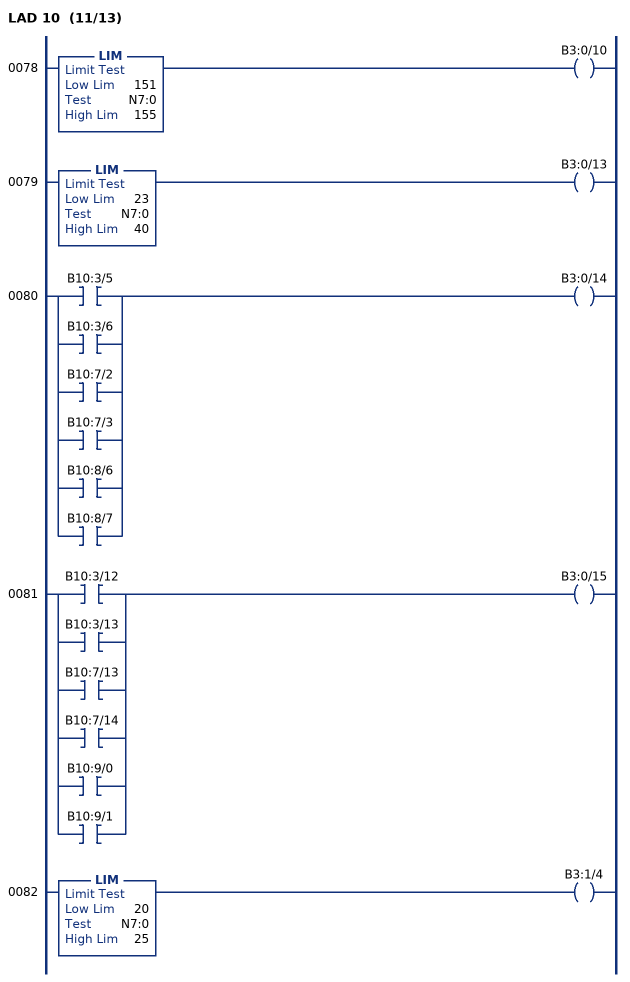
% Rung: 78 %
SOR LIM 151 N7:0 155 OTE B3:0/10 EOR
% Rung: 79 %
SOR LIM 23 N7:0 40 OTE B3:0/13 EOR
% Rung: 80 %
SOR BST XIC B10:3/5 NXB XIC B10:3/6 NXB XIC B10:7/2 NXB XIC B10:7/3 NXB XIC B10:8/6 NXB XIC B10:8/7 BND OTE B3:0/14 EOR
% Rung: 81 %
SOR BST XIC B10:3/12 NXB XIC B10:3/13 NXB XIC B10:7/13 NXB XIC B10:7/14 NXB XIC B10:9/0 NXB XIC B10:9/1 BND OTE B3:0/15 EOR
% Rung: 82 %
SOR LIM 20 N7:0 25 OTE B3:1/4 EOR

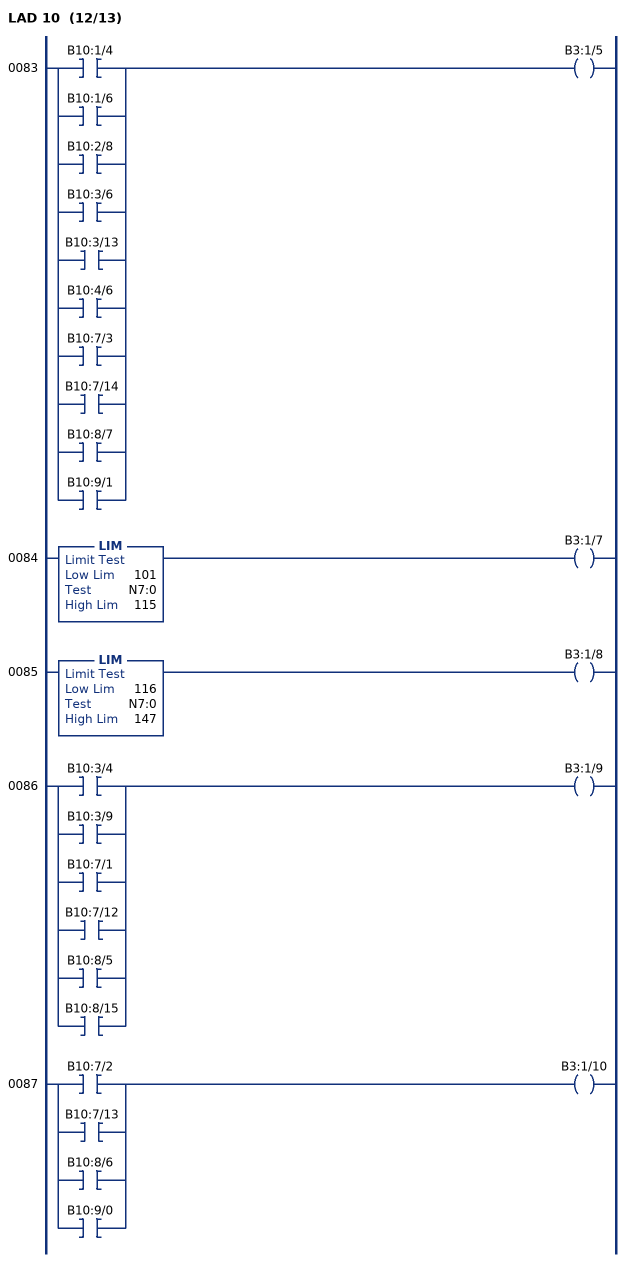
% Rung: 83 %
SOR BST XIC B10:1/4 NXB XIC B10:1/6 NXB XIC B10:2/8 NXB XIC B10:3/6 NXB XIC B10:3/13 NXB XIC B10:4/6 NXB XIC B10:7/3 NXB XIC B10:7/14 NXB XIC B10:8/7 NXB XIC B10:9/1 BND OTE B3:1/5 EOR
% Rung: 84 %
SOR LIM 101 N7:0 115 OTE B3:1/7 EOR
% Rung: 85 %
SOR LIM 116 N7:0 147 OTE B3:1/8 EOR
% Rung: 86 %
SOR BST XIC B10:3/4 NXB XIC B10:3/9 NXB XIC B10:7/1 NXB XIC B10:7/12 NXB XIC B10:8/5 NXB XIC B10:8/15 BND OTE B3:1/9 EOR
% Rung: 87 %
SOR BST XIC B10:7/2 NXB XIC B10:7/13 NXB XIC B10:8/6 NXB XIC B10:9/0 BND OTE B3:1/10 EOR

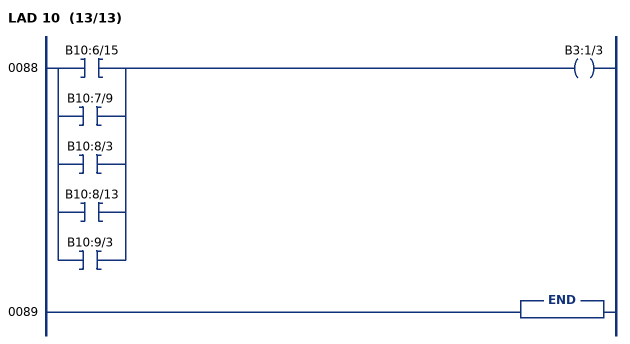
% Rung: 88 %
SOR BST XIC B10:6/15 NXB XIC B10:7/9 NXB XIC B10:8/3 NXB XIC B10:8/13 NXB XIC B10:9/3 BND OTE B3:1/3 EOR
% Rung: 89 %
SOR END EOR

LADDER 11
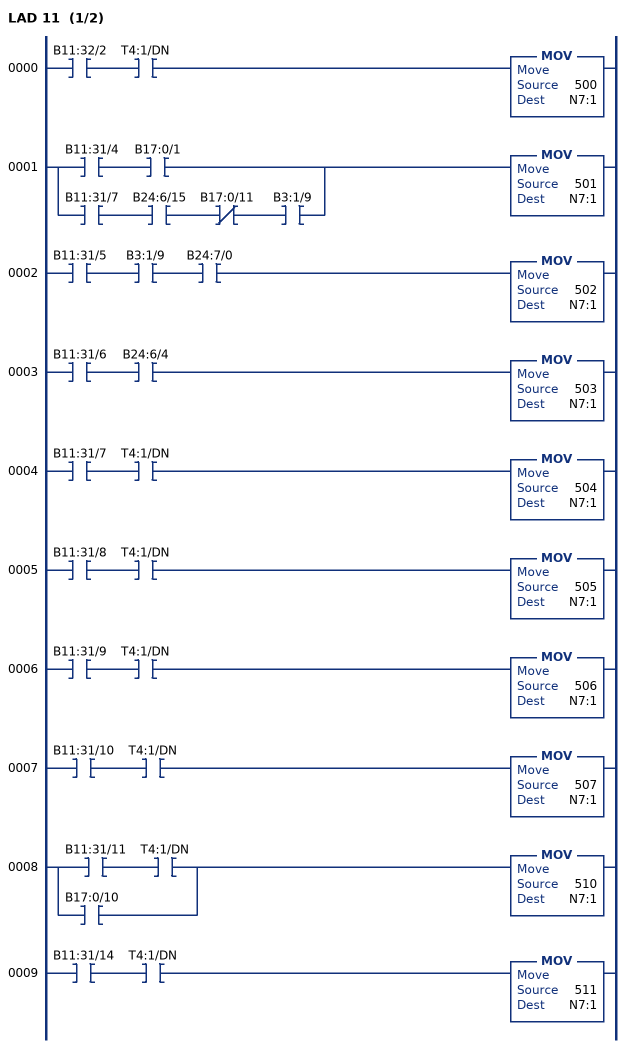
% Rung: 0 %
SOR XIC B11:32/2 XIC T4:1/DN MOV 500 N7:1 EOR
% Rung: 1 %
SOR BST XIC B11:31/4 XIC B17:0/1 NXB XIC B11:31/7 XIC B24:6/15 XIO B17:0/11 XIC B3:1/9 BND MOV 501 N7:1 EOR
% Rung: 2 %
SOR XIC B11:31/5 XIC B3:1/9 XIC B24:7/0 MOV 502 N7:1 EOR
% Rung: 3 %
SOR XIC B11:31/6 XIC B24:6/4 MOV 503 N7:1 EOR
% Rung: 4 %
SOR XIC B11:31/7 XIC T4:1/DN MOV 504 N7:1 EOR
% Rung: 5 %
SOR XIC B11:31/8 XIC T4:1/DN MOV 505 N7:1 EOR
% Rung: 6 %
SOR XIC B11:31/9 XIC T4:1/DN MOV 506 N7:1 EOR
% Rung: 7 %
SOR XIC B11:31/10 XIC T4:1/DN MOV 507 N7:1 EOR
% Rung: 8 %
SOR BST XIC B11:31/11 XIC T4:1/DN NXB XIC B17:0/10 BND MOV 510 N7:1 EOR
% Rung: 9 %
SOR XIC B11:31/14 XIC T4:1/DN MOV 511 N7:1 EOR

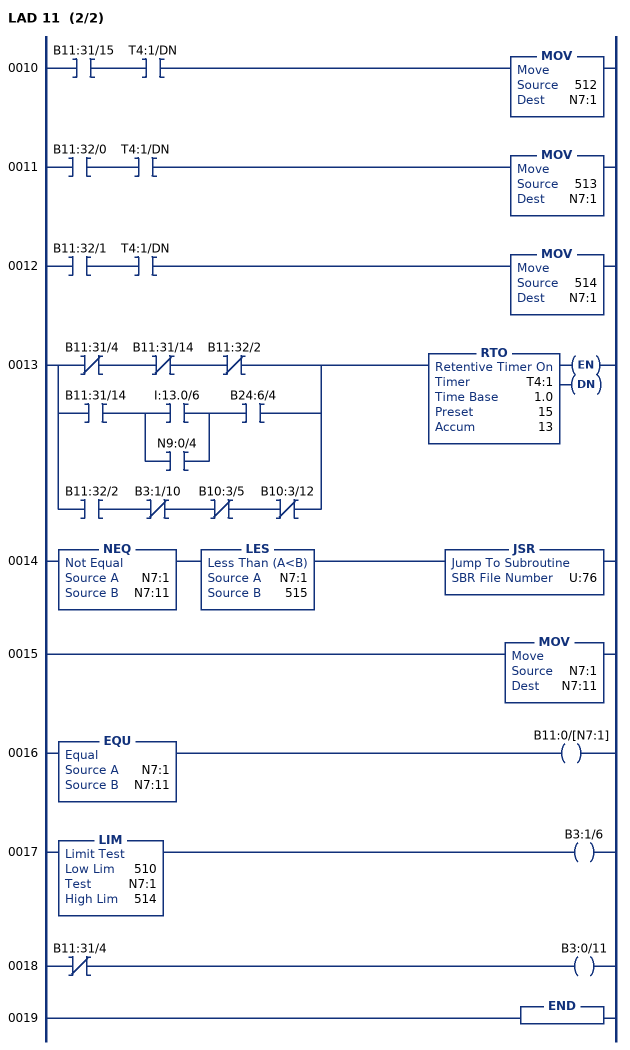
% Rung: 10 %
SOR XIC B11:31/15 XIC T4:1/DN MOV 512 N7:1 EOR
% Rung: 11 %
SOR XIC B11:32/0 XIC T4:1/DN MOV 513 N7:1 EOR
% Rung: 12 %
SOR XIC B11:32/1 XIC T4:1/DN MOV 514 N7:1 EOR
% Rung: 13 %
SOR BST XIO B11:31/4 XIO B11:31/14 XIO B11:32/2 NXB XIC B11:31/14 BST XIC I:13.0/6 NXB XIC N9:0/4 BND XIC B24:6/4 NXB XIC B11:32/2 XIO B3:1/10 XIO B10:3/5 XIO B10:3/12 BND RTO T4:1 1.0 15 13 EOR
% Rung: 14 %
SOR NEQ N7:1 N7:11 LES N7:1 515 JSR U:76 EOR
% Rung: 15 %
SOR MOV N7:1 N7:11 EOR
% Rung: 16 %
SOR EQU N7:1 N7:11 OTE B11:0/[N7:1] EOR
% Rung: 17 %
SOR LIM 510 N7:1 514 OTE B3:1/6 EOR
% Rung: 18 %
SOR XIO B11:31/4 OTE B3:0/11 EOR
% Rung: 19 %
SOR END EOR

LADDER 12
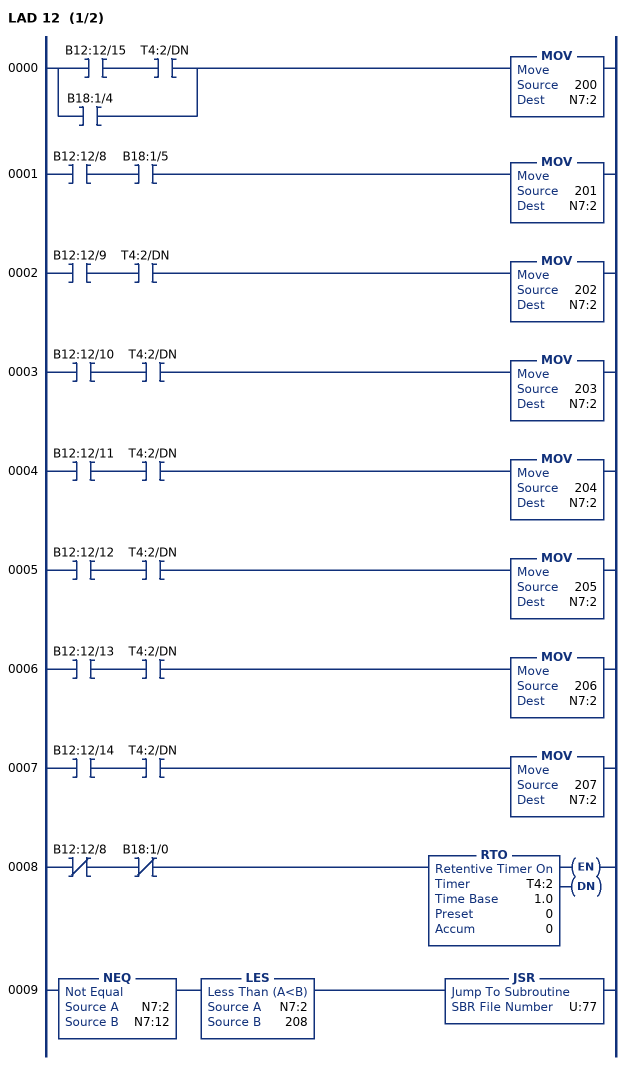
% Rung: 0 %
SOR BST XIC B12:12/15 XIC T4:2/DN NXB XIC B18:1/4 BND MOV 200 N7:2 EOR
% Rung: 1 %
SOR XIC B12:12/8 XIC B18:1/5 MOV 201 N7:2 EOR
% Rung: 2 %
SOR XIC B12:12/9 XIC T4:2/DN MOV 202 N7:2 EOR
% Rung: 3 %
SOR XIC B12:12/10 XIC T4:2/DN MOV 203 N7:2 EOR
% Rung: 4 %
SOR XIC B12:12/11 XIC T4:2/DN MOV 204 N7:2 EOR
% Rung: 5 %
SOR XIC B12:12/12 XIC T4:2/DN MOV 205 N7:2 EOR
% Rung: 6 %
SOR XIC B12:12/13 XIC T4:2/DN MOV 206 N7:2 EOR
% Rung: 7 %
SOR XIC B12:12/14 XIC T4:2/DN MOV 207 N7:2 EOR
% Rung: 8 %
SOR XIO B12:12/8 XIO B18:1/0 RTO T4:2 1.0 0 0 EOR
% Rung: 9 %
SOR NEQ N7:2 N7:12 LES N7:2 208 JSR U:77 EOR

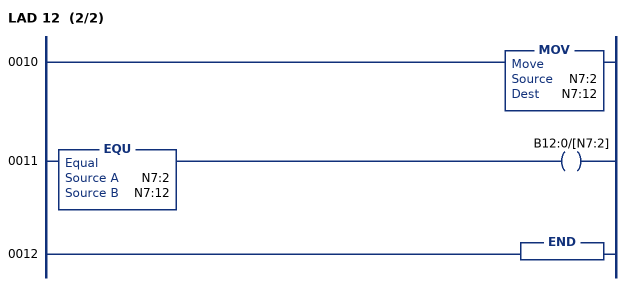
% Rung: 10 %
SOR MOV N7:2 N7:12 EOR
% Rung: 11 %
SOR EQU N7:2 N7:12 OTE B12:0/[N7:2] EOR
% Rung: 12 %
SOR END EOR

LADDER 15
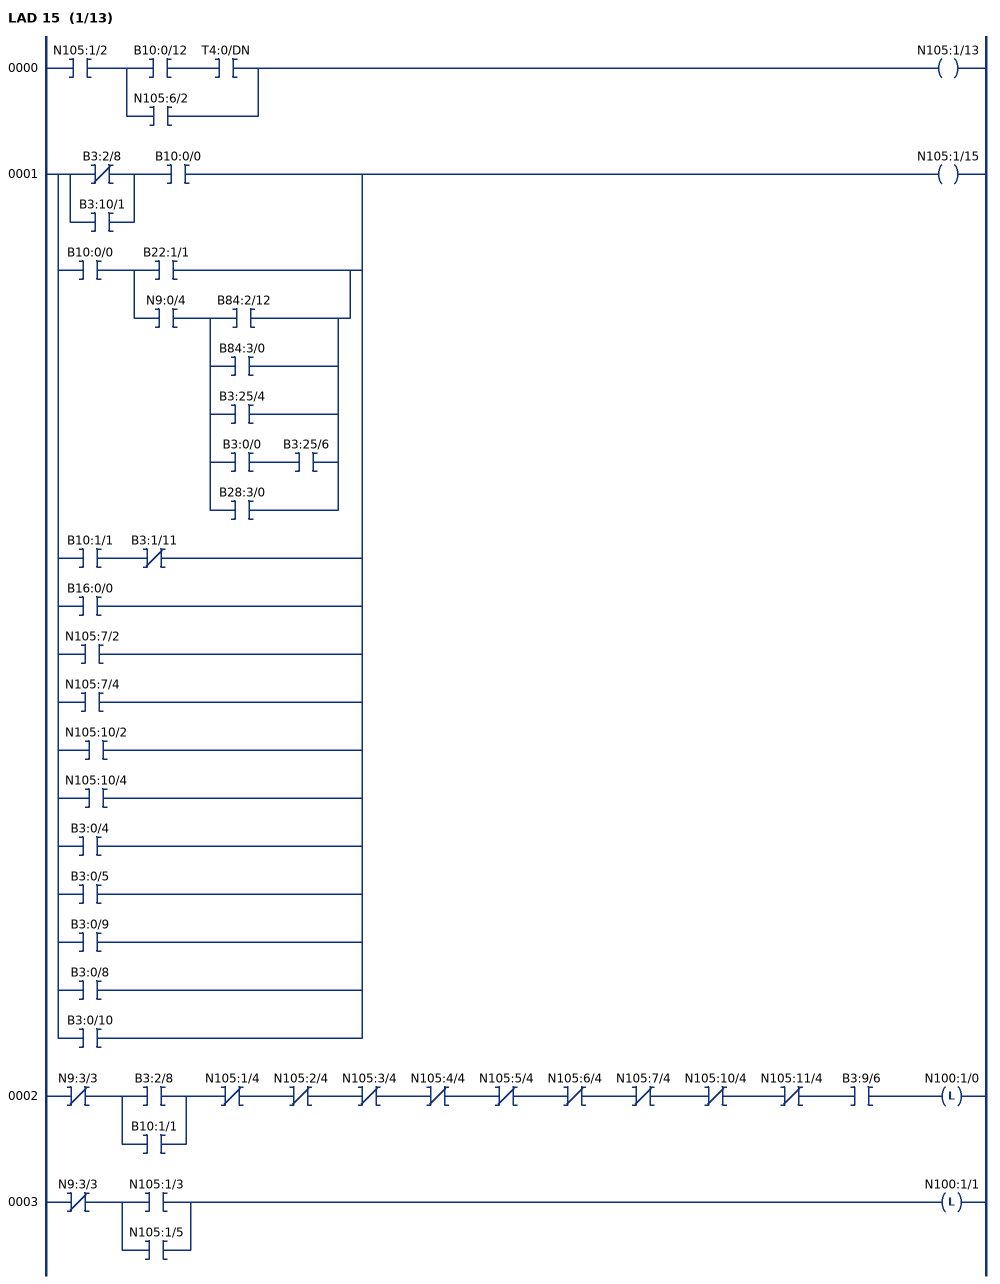
% Rung: 0 %
SOR XIC N105:1/2 BST XIC B10:0/12 XIC T4:0/DN NXB XIC N105:6/2 BND OTE N105:1/13 EOR
% Rung: 1 %
SOR BST BST XIO B3:2/8 NXB XIC B3:10/1 BND XIC B10:0/0 NXB XIC B10:0/0 BST XIC B22:1/1 NXB XIC N9:0/4 BST XIC B84:2/12 NXB XIC B84:3/0 NXB XIC B3:25/4 NXB XIC B3:0/0 XIC B3:25/6 NXB XIC B28:3/0 BND BND NXB XIC B10:1/1 XIO B3:1/11 NXB XIC B16:0/0 NXB XIC N105:7/2 NXB XIC N105:7/4 NXB XIC N105:10/2 NXB XIC N105:10/4 NXB XIC B3:0/4 NXB XIC B3:0/5 NXB XIC B3:0/9 NXB XIC B3:0/8 NXB XIC B3:0/10 BND OTE N105:1/15 EOR
% Rung: 2 %
SOR XIO N9:3/3 BST XIC B3:2/8 NXB XIC B10:1/1 BND XIO N105:1/4 XIO N105:2/4 XIO N105:3/4 XIO N105:4/4 XIO N105:5/4 XIO N105:6/4 XIO N105:7/4 XIO N105:10/4 XIO N105:11/4 XIC B3:9/6 OTL N100:1/0 EOR
% Rung: 3 %
SOR XIO N9:3/3 BST XIC N105:1/3 NXB XIC N105:1/5 BND OTL N100:1/1 EOR

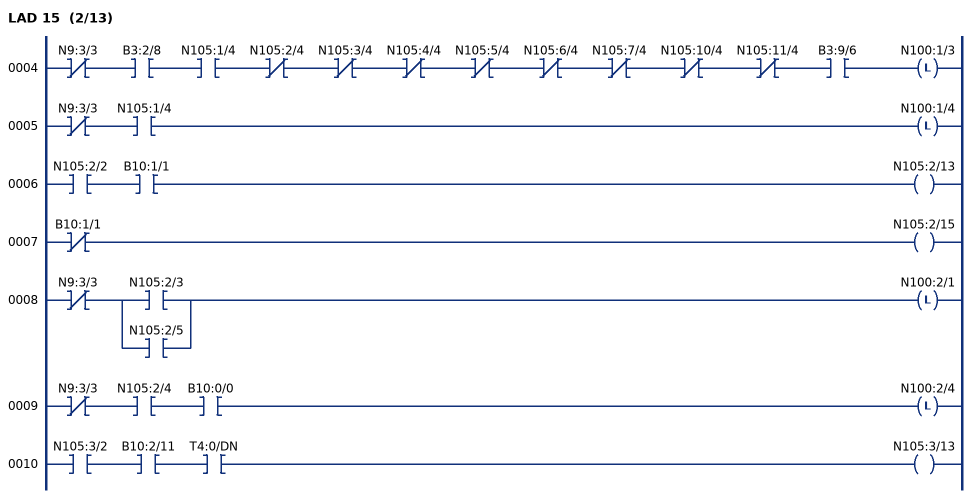
% Rung: 4 %
SOR XIO N9:3/3 XIC B3:2/8 XIC N105:1/4 XIO N105:2/4 XIO N105:3/4 XIO N105:4/4 XIO N105:5/4 XIO N105:6/4 XIO N105:7/4 XIO N105:10/4 XIO N105:11/4 XIC B3:9/6 OTL N100:1/3 EOR
% Rung: 5 %
SOR XIO N9:3/3 XIC N105:1/4 OTL N100:1/4 EOR
% Rung: 6 %
SOR XIC N105:2/2 XIC B10:1/1 OTE N105:2/13 EOR
% Rung: 7 %
SOR XIO B10:1/1 OTE N105:2/15 EOR
% Rung: 8 %
SOR XIO N9:3/3 BST XIC N105:2/3 NXB XIC N105:2/5 BND OTL N100:2/1 EOR
% Rung: 9 %
SOR XIO N9:3/3 XIC N105:2/4 XIC B10:0/0 OTL N100:2/4 EOR
% Rung: 10 %
SOR XIC N105:3/2 XIC B10:2/11 XIC T4:0/DN OTE N105:3/13 EOR

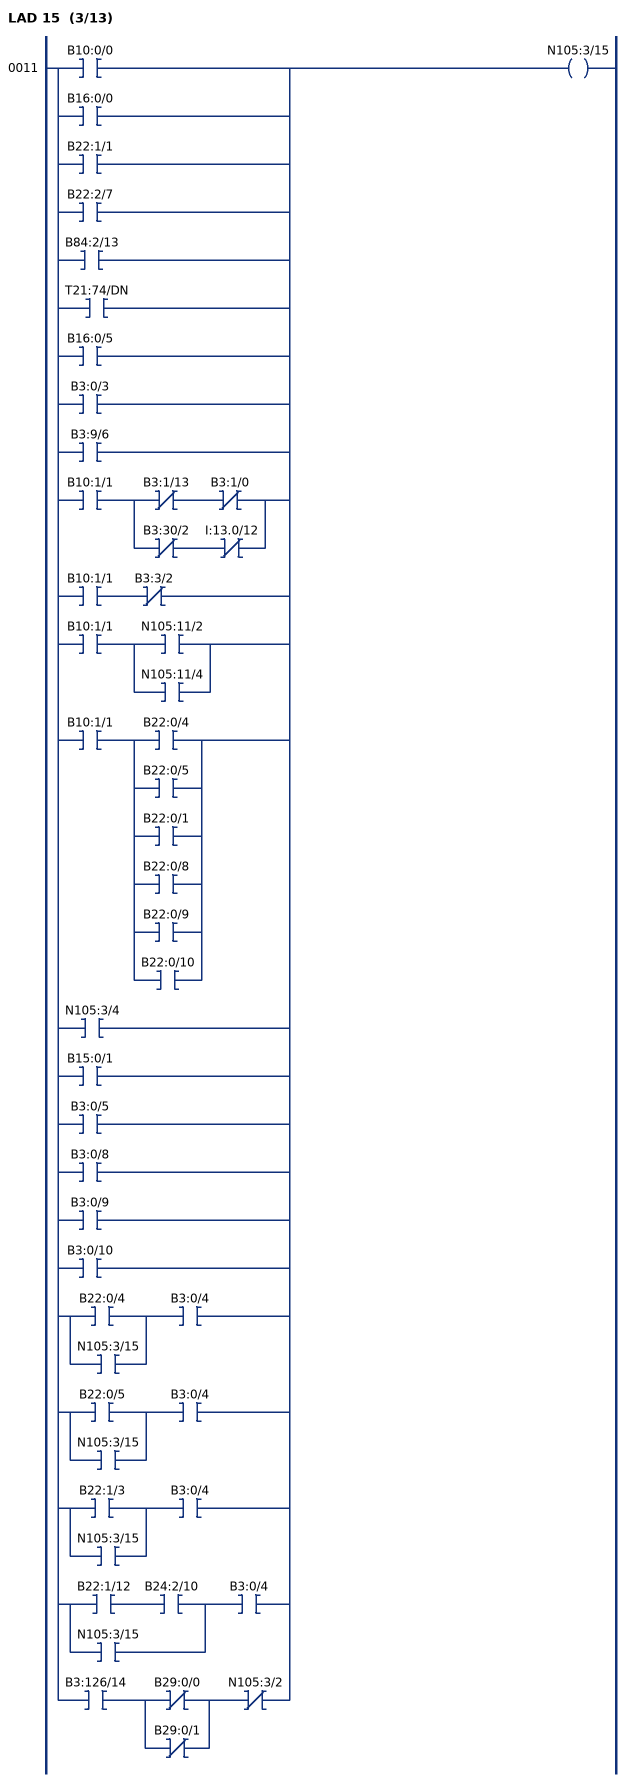
% Rung: 11 %
SOR BST XIC B10:0/0 NXB XIC B16:0/0 NXB XIC B22:1/1 NXB XIC B22:2/7 NXB XIC B84:2/13 NXB XIC T21:74/DN NXB XIC B16:0/5 NXB XIC B3:0/3 NXB XIC B3:9/6 NXB XIC B10:1/1 BST XIO B3:1/13 XIO B3:1/0 NXB XIO B3:30/2 XIO I:13.0/12 BND NXB XIC B10:1/1 XIO B3:3/2 NXB XIC B10:1/1 BST XIC N105:11/2 NXB XIC N105:11/4 BND NXB XIC B10:1/1 BST XIC B22:0/4 NXB XIC B22:0/5 NXB XIC B22:0/1 NXB XIC B22:0/8 NXB XIC B22:0/9 NXB XIC B22:0/10 BND NXB XIC N105:3/4 NXB XIC B15:0/1 NXB XIC B3:0/5 NXB XIC B3:0/8 NXB XIC B3:0/9 NXB XIC B3:0/10 NXB BST XIC B22:0/4 NXB XIC N105:3/15 BND XIC B3:0/4 NXB BST XIC B22:0/5 NXB XIC N105:3/15 BND XIC B3:0/4 NXB BST XIC B22:1/3 NXB XIC N105:3/15 BND XIC B3:0/4 NXB BST XIC B22:1/12 XIC B24:2/10 NXB XIC N105:3/15 BND XIC B3:0/4 NXB XIC B3:126/14 BST XIO B29:0/0 NXB XIO B29:0/1 BND XIO N105:3/2 BND OTE N105:3/15 EOR

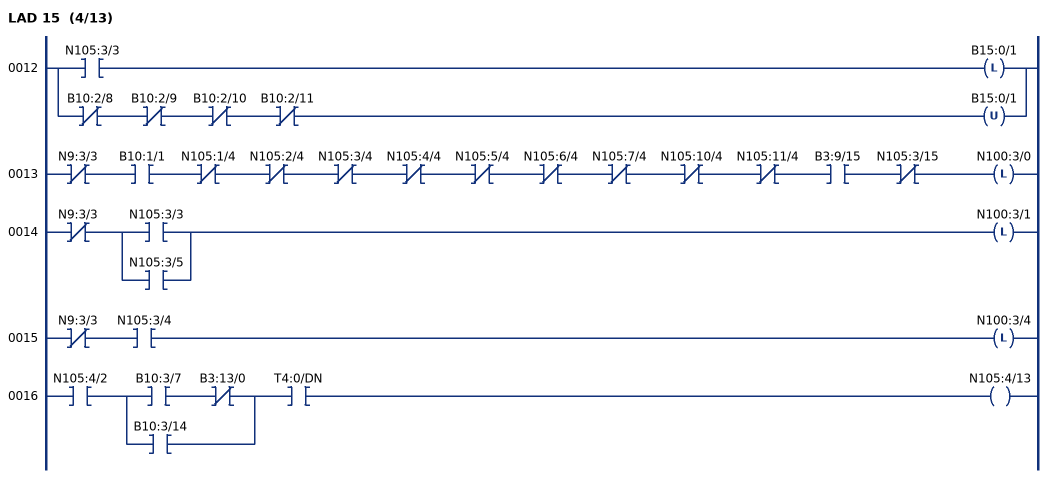
% Rung: 12 %
SOR BST XIC N105:3/3 OTL B15:0/1 NXB XIO B10:2/8 XIO B10:2/9 XIO B10:2/10 XIO B10:2/11 OTU B15:0/1 BND EOR
% Rung: 13 %
SOR XIO N9:3/3 XIC B10:1/1 XIO N105:1/4 XIO N105:2/4 XIO N105:3/4 XIO N105:4/4 XIO N105:5/4 XIO N105:6/4 XIO N105:7/4 XIO N105:10/4 XIO N105:11/4 XIC B3:9/15 XIO N105:3/15 OTL N100:3/0 EOR
% Rung: 14 %
SOR XIO N9:3/3 BST XIC N105:3/3 NXB XIC N105:3/5 BND OTL N100:3/1 EOR
% Rung: 15 %
SOR XIO N9:3/3 XIC N105:3/4 OTL N100:3/4 EOR
% Rung: 16 %
SOR XIC N105:4/2 BST XIC B10:3/7 XIO B3:13/0 NXB XIC B10:3/14 BND XIC T4:0/DN OTE N105:4/13 EOR

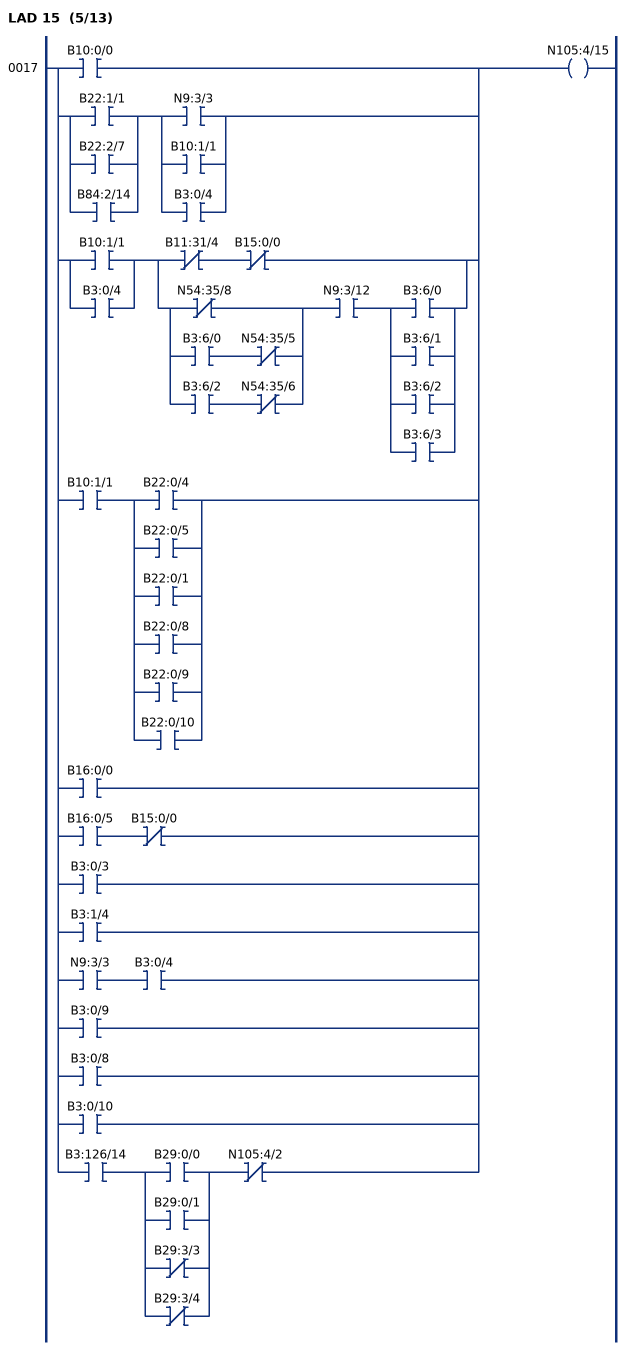
% Rung: 17 %
SOR BST XIC B10:0/0 NXB BST XIC B22:1/1 NXB XIC B22:2/7 NXB XIC B84:2/14 BND BST XIC N9:3/3 NXB XIC B10:1/1 NXB XIC B3:0/4 BND NXB BST XIC B10:1/1 NXB XIC B3:0/4 BND BST XIO B11:31/4 XIO B15:0/0 NXB BST XIO N54:35/8 NXB XIC B3:6/0 XIO N54:35/5 NXB XIC B3:6/2 XIO N54:35/6 BND XIC N9:3/12 BST XIC B3:6/0 NXB XIC B3:6/1 NXB XIC B3:6/2 NXB XIC B3:6/3 BND BND NXB XIC B10:1/1 BST XIC B22:0/4 NXB XIC B22:0/5 NXB XIC B22:0/1 NXB XIC B22:0/8 NXB XIC B22:0/9 NXB XIC B22:0/10 BND NXB XIC B16:0/0 NXB XIC B16:0/5 XIO B15:0/0 NXB XIC B3:0/3 NXB XIC B3:1/4 NXB XIC N9:3/3 XIC B3:0/4 NXB XIC B3:0/9 NXB XIC B3:0/8 NXB XIC B3:0/10 NXB XIC B3:126/14 BST XIC B29:0/0 NXB XIC B29:0/1 NXB XIO B29:3/3 NXB XIO B29:3/4 BND XIO N105:4/2 BND OTE N105:4/15 EOR

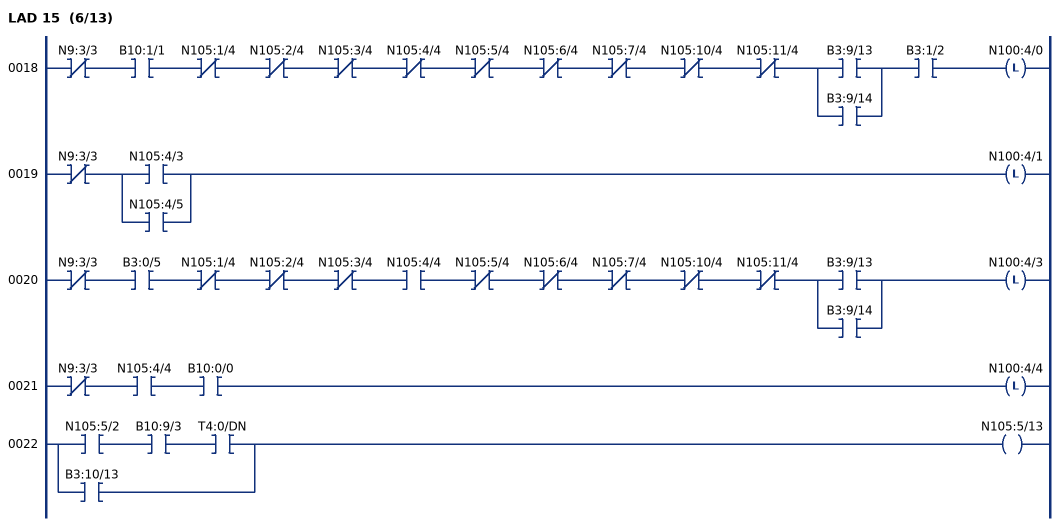
% Rung: 18 %
SOR XIO N9:3/3 XIC B10:1/1 XIO N105:1/4 XIO N105:2/4 XIO N105:3/4 XIO N105:4/4 XIO N105:5/4 XIO N105:6/4 XIO N105:7/4 XIO N105:10/4 XIO N105:11/4 BST XIC B3:9/13 NXB XIC B3:9/14 BND XIC B3:1/2 OTL N100:4/0 EOR
% Rung: 19 %
SOR XIO N9:3/3 BST XIC N105:4/3 NXB XIC N105:4/5 BND OTL N100:4/1 EOR
% Rung: 20 %
SOR XIO N9:3/3 XIC B3:0/5 XIO N105:1/4 XIO N105:2/4 XIO N105:3/4 XIC N105:4/4 XIO N105:5/4 XIO N105:6/4 XIO N105:7/4 XIO N105:10/4 XIO N105:11/4 BST XIC B3:9/13 NXB XIC B3:9/14 BND OTL N100:4/3 EOR
% Rung: 21 %
SOR XIO N9:3/3 XIC N105:4/4 XIC B10:0/0 OTL N100:4/4 EOR
% Rung: 22 %
SOR BST XIC N105:5/2 XIC B10:9/3 XIC T4:0/DN NXB XIC B3:10/13 BND OTE N105:5/13 EOR

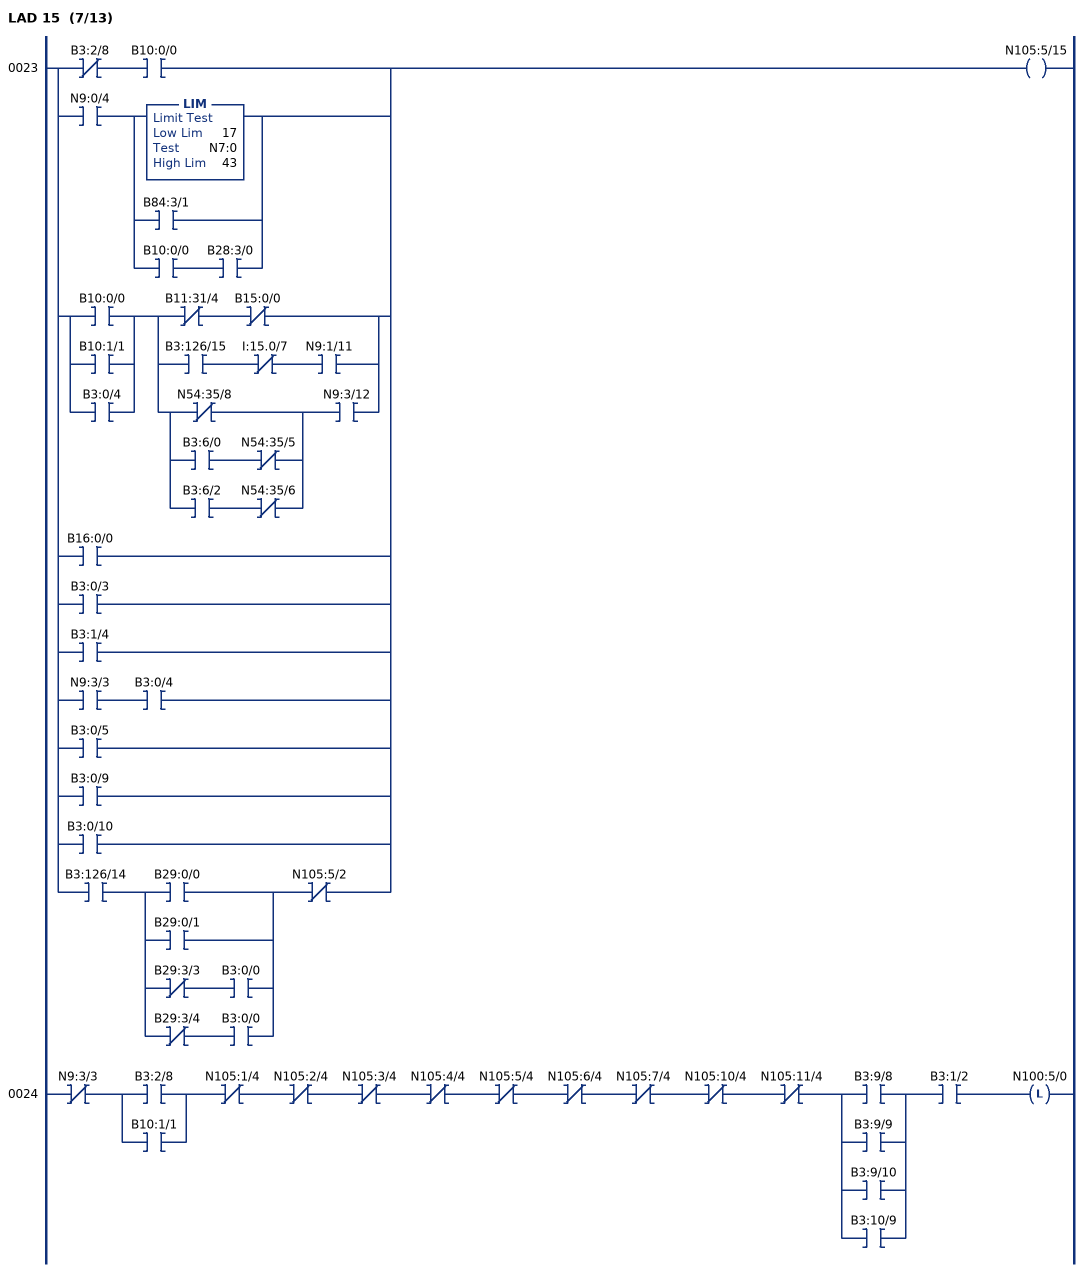
% Rung: 23 %
SOR BST XIO B3:2/8 XIC B10:0/0 NXB XIC N9:0/4 BST LIM 17 N7:0 43 NXB XIC B84:3/1 NXB XIC B10:0/0 XIC B28:3/0 BND NXB BST XIC B10:0/0 NXB XIC B10:1/1 NXB XIC B3:0/4 BND BST XIO B11:31/4 XIO B15:0/0 NXB XIC B3:126/15 XIO I:15.0/7 XIC N9:1/11 NXB BST XIO N54:35/8 NXB XIC B3:6/0 XIO N54:35/5 NXB XIC B3:6/2 XIO N54:35/6 BND XIC N9:3/12 BND NXB XIC B16:0/0 NXB XIC B3:0/3 NXB XIC B3:1/4 NXB XIC N9:3/3 XIC B3:0/4 NXB XIC B3:0/5 NXB XIC B3:0/9 NXB XIC B3:0/10 NXB XIC B3:126/14 BST XIC B29:0/0 NXB XIC B29:0/1 NXB XIO B29:3/3 XIC B3:0/0 NXB XIO B29:3/4 XIC B3:0/0 BND XIO N105:5/2 BND OTE N105:5/15 EOR
% Rung: 24 %
SOR XIO N9:3/3 BST XIC B3:2/8 NXB XIC B10:1/1 BND XIO N105:1/4 XIO N105:2/4 XIO N105:3/4 XIO N105:4/4 XIO N105:5/4 XIO N105:6/4 XIO N105:7/4 XIO N105:10/4 XIO N105:11/4 BST XIC B3:9/8 NXB XIC B3:9/9 NXB XIC B3:9/10 NXB XIC B3:10/9 BND XIC B3:1/2 OTL N100:5/0 EOR

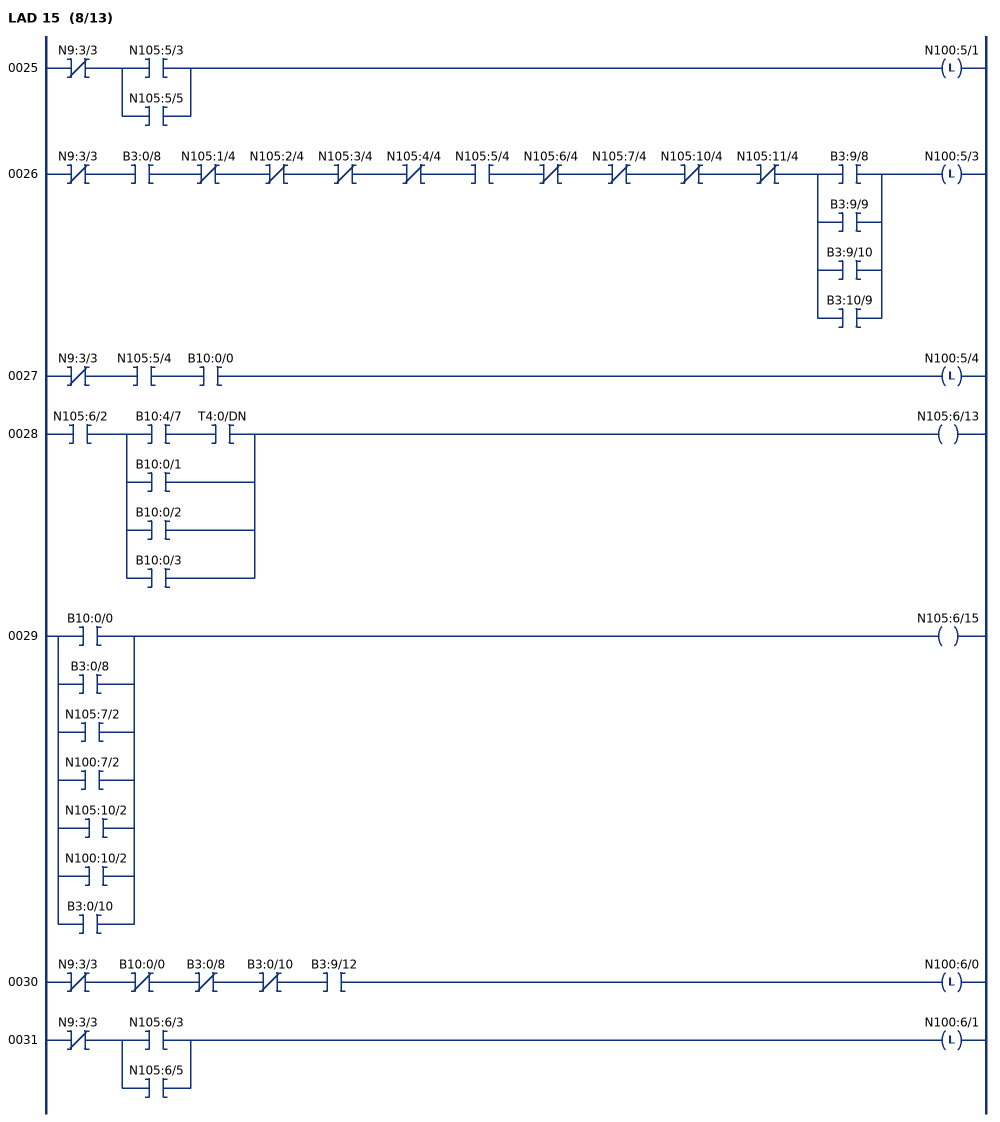
% Rung: 25 %
SOR XIO N9:3/3 BST XIC N105:5/3 NXB XIC N105:5/5 BND OTL N100:5/1 EOR
% Rung: 26 %
SOR XIO N9:3/3 XIC B3:0/8 XIO N105:1/4 XIO N105:2/4 XIO N105:3/4 XIO N105:4/4 XIC N105:5/4 XIO N105:6/4 XIO N105:7/4 XIO N105:10/4 XIO N105:11/4 BST XIC B3:9/8 NXB XIC B3:9/9 NXB XIC B3:9/10 NXB XIC B3:10/9 BND OTL N100:5/3 EOR
% Rung: 27 %
SOR XIO N9:3/3 XIC N105:5/4 XIC B10:0/0 OTL N100:5/4 EOR
% Rung: 28 %
SOR XIC N105:6/2 BST XIC B10:4/7 XIC T4:0/DN NXB XIC B10:0/1 NXB XIC B10:0/2 NXB XIC B10:0/3 BND OTE N105:6/13 EOR
% Rung: 29 %
SOR BST XIC B10:0/0 NXB XIC B3:0/8 NXB BST XIC N105:7/2 NXB XIC N100:7/2 NXB XIC N105:10/2 NXB XIC N100:10/2 BND NXB XIC B3:0/10 BND OTE N105:6/15 EOR
% Rung: 30 %
SOR XIO N9:3/3 XIO B10:0/0 XIO B3:0/8 XIO B3:0/10 XIC B3:9/12 OTL N100:6/0 EOR
% Rung: 31 %
SOR XIO N9:3/3 BST XIC N105:6/3 NXB XIC N105:6/5 BND OTL N100:6/1 EOR

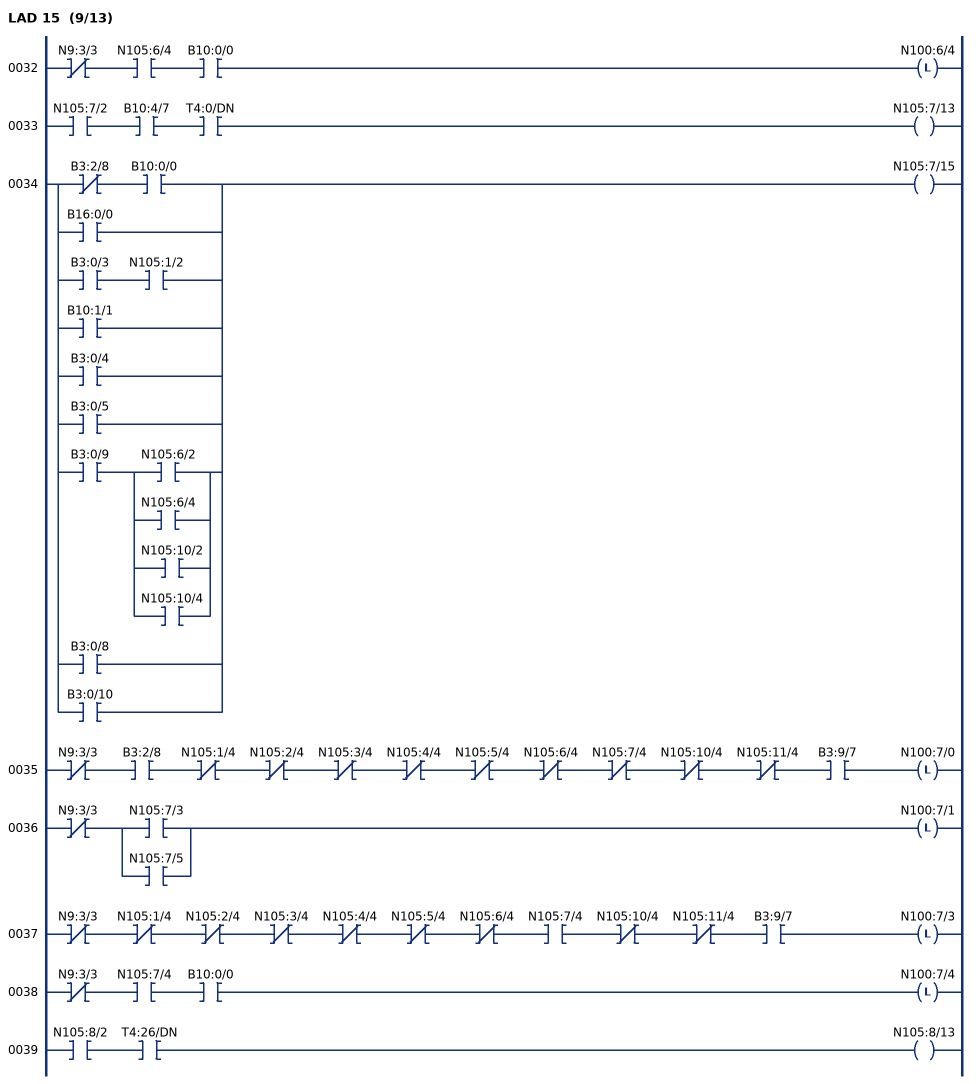
% Rung: 32 %
SOR XIO N9:3/3 XIC N105:6/4 XIC B10:0/0 OTL N100:6/4 EOR
% Rung: 33 %
SOR XIC N105:7/2 XIC B10:4/7 XIC T4:0/DN OTE N105:7/13 EOR
% Rung: 34 %
SOR BST XIO B3:2/8 XIC B10:0/0 NXB XIC B16:0/0 NXB XIC B3:0/3 XIC N105:1/2 NXB XIC B10:1/1 NXB XIC B3:0/4 NXB XIC B3:0/5 NXB XIC B3:0/9 BST XIC N105:6/2 NXB XIC N105:6/4 NXB XIC N105:10/2 NXB XIC N105:10/4 BND NXB XIC B3:0/8 NXB XIC B3:0/10 BND OTE N105:7/15 EOR
% Rung: 35 %
SOR XIO N9:3/3 XIC B3:2/8 XIO N105:1/4 XIO N105:2/4 XIO N105:3/4 XIO N105:4/4 XIO N105:5/4 XIO N105:6/4 XIO N105:7/4 XIO N105:10/4 XIO N105:11/4 XIC B3:9/7 OTL N100:7/0 EOR
% Rung: 36 %
SOR XIO N9:3/3 BST XIC N105:7/3 NXB XIC N105:7/5 BND OTL N100:7/1 EOR
% Rung: 37 %
SOR XIO N9:3/3 XIO N105:1/4 XIO N105:2/4 XIO N105:3/4 XIO N105:4/4 XIO N105:5/4 XIO N105:6/4 XIC N105:7/4 XIO N105:10/4 XIO N105:11/4 XIC B3:9/7 OTL N100:7/3 EOR
% Rung: 38 %
SOR XIO N9:3/3 XIC N105:7/4 XIC B10:0/0 OTL N100:7/4 EOR
% Rung: 39 %
SOR XIC N105:8/2 XIC T4:26/DN OTE N105:8/13 EOR

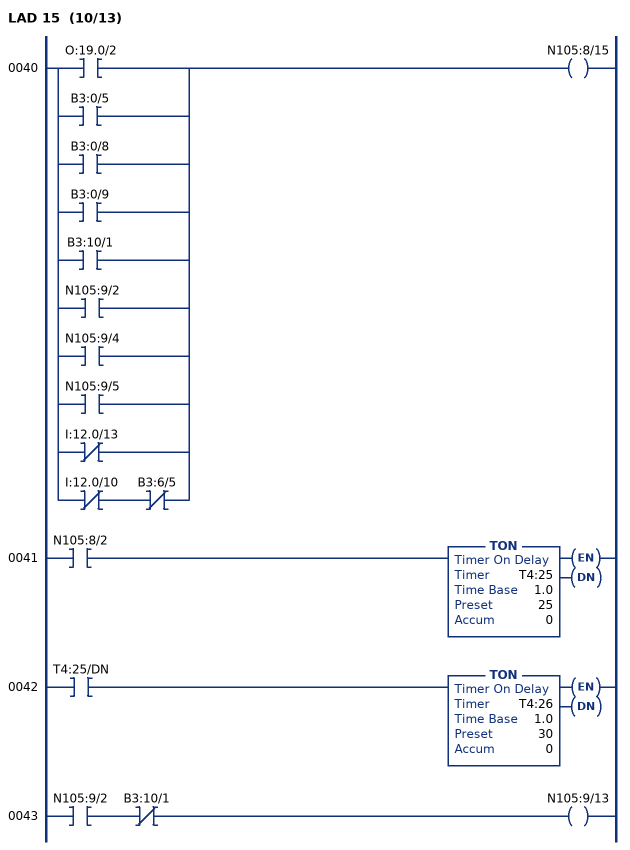
% Rung: 40 %
SOR BST XIC O:19.0/2 NXB XIC B3:0/5 NXB XIC B3:0/8 NXB XIC B3:0/9 NXB XIC B3:10/1 NXB XIC N105:9/2 NXB XIC N105:9/4 NXB XIC N105:9/5 NXB XIO I:12.0/13 NXB XIO I:12.0/10 XIO B3:6/5 BND OTE N105:8/15 EOR
% Rung: 41 %
SOR XIC N105:8/2 TON T4:25 1.0 25 0 EOR
% Rung: 42 %
SOR XIC T4:25/DN TON T4:26 1.0 30 0 EOR
% Rung: 43 %
SOR XIC N105:9/2 XIO B3:10/1 OTE N105:9/13 EOR

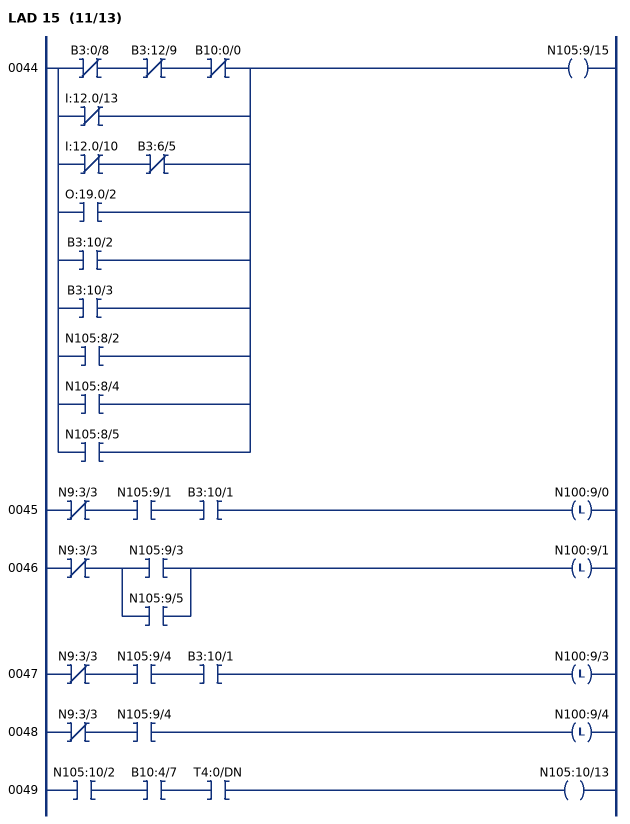
% Rung: 44 %
SOR BST XIO B3:0/8 XIO B3:12/9 XIO B10:0/0 NXB XIO I:12.0/13 NXB XIO I:12.0/10 XIO B3:6/5 NXB XIC O:19.0/2 NXB XIC B3:10/2 NXB XIC B3:10/3 NXB XIC N105:8/2 NXB XIC N105:8/4 NXB XIC N105:8/5 BND OTE N105:9/15 EOR
% Rung: 45 %
SOR XIO N9:3/3 XIC N105:9/1 XIC B3:10/1 OTL N100:9/0 EOR
% Rung: 46 %
SOR XIO N9:3/3 BST XIC N105:9/3 NXB XIC N105:9/5 BND OTL N100:9/1 EOR
% Rung: 47 %
SOR XIO N9:3/3 XIC N105:9/4 XIC B3:10/1 OTL N100:9/3 EOR
% Rung: 48 %
SOR XIO N9:3/3 XIC N105:9/4 OTL N100:9/4 EOR
% Rung: 49 %
SOR XIC N105:10/2 XIC B10:4/7 XIC T4:0/DN OTE N105:10/13 EOR

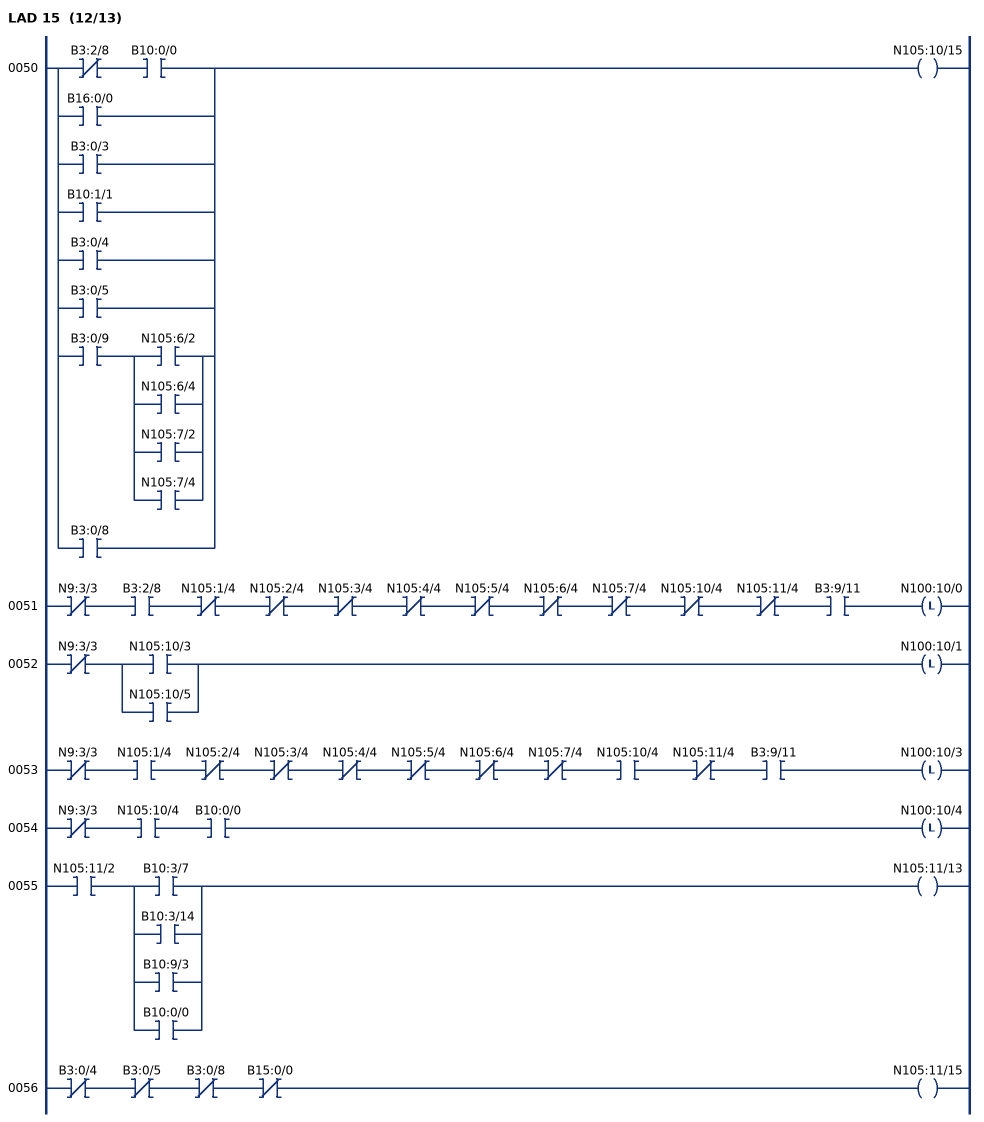
% Rung: 50 %
SOR BST XIO B3:2/8 XIC B10:0/0 NXB XIC B16:0/0 NXB XIC B3:0/3 NXB XIC B10:1/1 NXB XIC B3:0/4 NXB XIC B3:0/5 NXB XIC B3:0/9 BST XIC N105:6/2 NXB XIC N105:6/4 NXB XIC N105:7/2 NXB XIC N105:7/4 BND NXB XIC B3:0/8 BND OTE N105:10/15 EOR
% Rung: 51 %
SOR XIO N9:3/3 XIC B3:2/8 XIO N105:1/4 XIO N105:2/4 XIO N105:3/4 XIO N105:4/4 XIO N105:5/4 XIO N105:6/4 XIO N105:7/4 XIO N105:10/4 XIO N105:11/4 XIC B3:9/11 OTL N100:10/0 EOR
% Rung: 52 %
SOR XIO N9:3/3 BST XIC N105:10/3 NXB XIC N105:10/5 BND OTL N100:10/1 EOR
% Rung: 53 %
SOR XIO N9:3/3 XIC N105:1/4 XIO N105:2/4 XIO N105:3/4 XIO N105:4/4 XIO N105:5/4 XIO N105:6/4 XIO N105:7/4 XIC N105:10/4 XIO N105:11/4 XIC B3:9/11 OTL N100:10/3 EOR
% Rung: 54 %
SOR XIO N9:3/3 XIC N105:10/4 XIC B10:0/0 OTL N100:10/4 EOR
% Rung: 55 %
SOR XIC N105:11/2 BST XIC B10:3/7 NXB XIC B10:3/14 NXB XIC B10:9/3 NXB XIC B10:0/0 BND OTE N105:11/13 EOR
% Rung: 56 %
SOR XIO B3:0/4 XIO B3:0/5 XIO B3:0/8 XIO B15:0/0 OTE N105:11/15 EOR

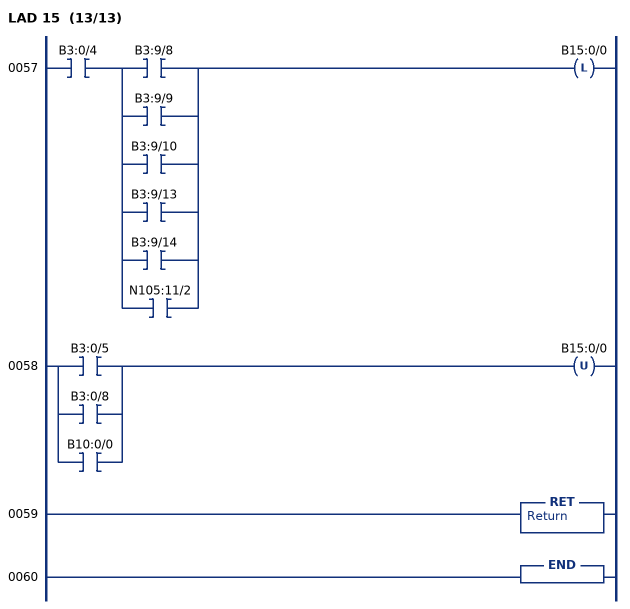
% Rung: 57 %
SOR XIC B3:0/4 BST XIC B3:9/8 NXB XIC B3:9/9 NXB XIC B3:9/10 NXB XIC B3:9/13 NXB XIC B3:9/14 NXB XIC N105:11/2 BND OTL B15:0/0 EOR
% Rung: 58 %
SOR BST XIC B3:0/5 NXB XIC B3:0/8 NXB XIC B10:0/0 BND OTU B15:0/0 EOR
% Rung: 59 %
SOR RET EOR
% Rung: 60 %
SOR END EOR

LADDER 16
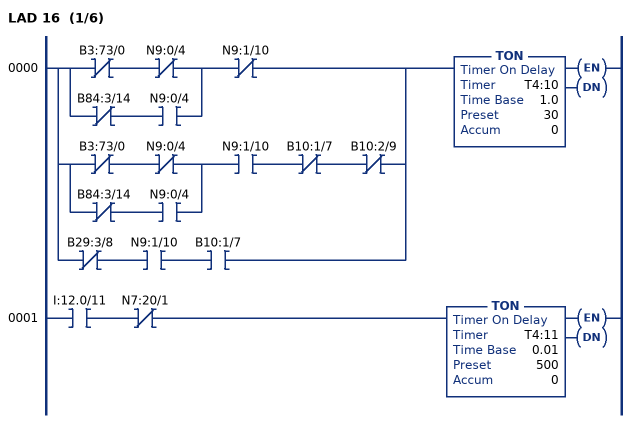
% Rung: 0 %
SOR BST BST XIO B3:73/0 XIO N9:0/4 NXB XIO B84:3/14 XIC N9:0/4 BND XIO N9:1/10 NXB BST XIO B3:73/0 XIO N9:0/4 NXB XIO B84:3/14 XIC N9:0/4 BND XIC N9:1/10 XIO B10:1/7 XIO B10:2/9 NXB XIO B29:3/8 XIC N9:1/10 XIC B10:1/7 BND TON T4:10 1.0 30 0 EOR
% Rung: 1 %
SOR XIC I:12.0/11 XIO N7:20/1 TON T4:11 0.01 500 0 EOR

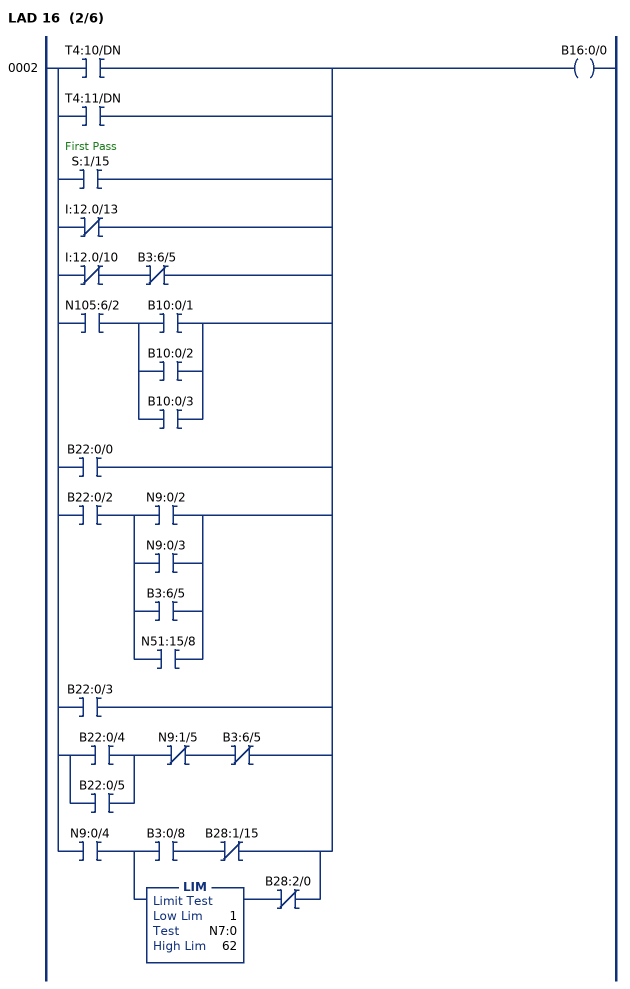
% Rung: 2 %
SOR BST XIC T4:10/DN NXB XIC T4:11/DN NXB XIC S:1/15 NXB XIO I:12.0/13 NXB XIO I:12.0/10 XIO B3:6/5 NXB XIC N105:6/2 BST XIC B10:0/1 NXB XIC B10:0/2 NXB XIC B10:0/3 BND NXB XIC B22:0/0 NXB XIC B22:0/2 BST XIC N9:0/2 NXB XIC N9:0/3 NXB XIC B3:6/5 NXB XIC N51:15/8 BND NXB XIC B22:0/3 NXB BST XIC B22:0/4 NXB XIC B22:0/5 BND XIO N9:1/5 XIO B3:6/5 NXB XIC N9:0/4 BST XIC B3:0/8 XIO B28:1/15 NXB LIM 1 N7:0 62 XIO B28:2/0 BND BND OTE B16:0/0 EOR
%   S:1/15  "First Pass" %

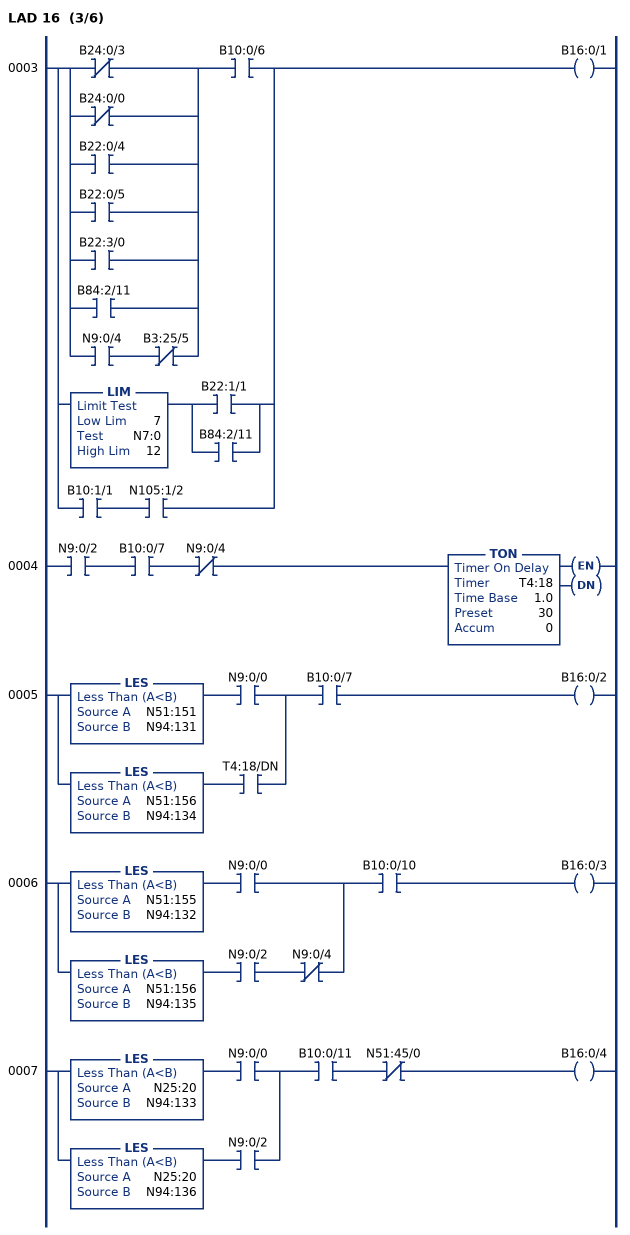
% Rung: 3 %
SOR BST BST XIO B24:0/3 NXB XIO B24:0/0 NXB XIC B22:0/4 NXB XIC B22:0/5 NXB XIC B22:3/0 NXB XIC B84:2/11 NXB XIC N9:0/4 XIO B3:25/5 BND XIC B10:0/6 NXB LIM 7 N7:0 12 BST XIC B22:1/1 NXB XIC B84:2/11 BND NXB XIC B10:1/1 XIC N105:1/2 BND OTE B16:0/1 EOR
% Rung: 4 %
SOR XIC N9:0/2 XIC B10:0/7 XIO N9:0/4 TON T4:18 1.0 30 0 EOR
% Rung: 5 %
SOR BST LES N51:151 N94:131 XIC N9:0/0 NXB LES N51:156 N94:134 XIC T4:18/DN BND XIC B10:0/7 OTE B16:0/2 EOR
% Rung: 6 %
SOR BST LES N51:155 N94:132 XIC N9:0/0 NXB LES N51:156 N94:135 XIC N9:0/2 XIO N9:0/4 BND XIC B10:0/10 OTE B16:0/3 EOR
% Rung: 7 %
SOR BST LES N25:20 N94:133 XIC N9:0/0 NXB LES N25:20 N94:136 XIC N9:0/2 BND XIC B10:0/11 XIO N51:45/0 OTE B16:0/4 EOR

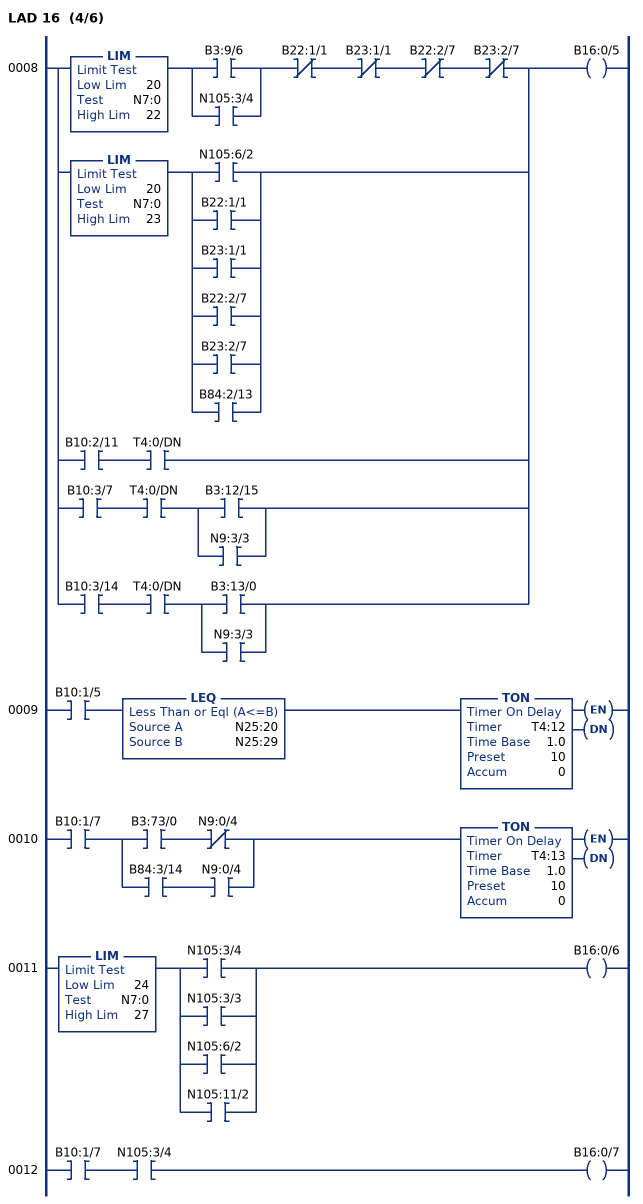
% Rung: 8 %
SOR BST LIM 20 N7:0 22 BST XIC B3:9/6 NXB XIC N105:3/4 BND XIO B22:1/1 XIO B23:1/1 XIO B22:2/7 XIO B23:2/7 NXB LIM 20 N7:0 23 BST XIC N105:6/2 NXB XIC B22:1/1 NXB XIC B23:1/1 NXB XIC B22:2/7 NXB XIC B23:2/7 NXB XIC B84:2/13 BND NXB XIC B10:2/11 XIC T4:0/DN NXB XIC B10:3/7 XIC T4:0/DN BST XIC B3:12/15 NXB XIC N9:3/3 BND NXB XIC B10:3/14 XIC T4:0/DN BST XIC B3:13/0 NXB XIC N9:3/3 BND BND OTE B16:0/5 EOR
% Rung: 9 %
SOR XIC B10:1/5 LEQ N25:20 N25:29 TON T4:12 1.0 10 0 EOR
% Rung: 10 %
SOR XIC B10:1/7 BST XIC B3:73/0 XIO N9:0/4 NXB XIC B84:3/14 XIC N9:0/4 BND TON T4:13 1.0 10 0 EOR
% Rung: 11 %
SOR LIM 24 N7:0 27 BST XIC N105:3/4 NXB XIC N105:3/3 NXB XIC N105:6/2 NXB XIC N105:11/2 BND OTE B16:0/6 EOR
% Rung: 12 %
SOR XIC B10:1/7 XIC N105:3/4 OTE B16:0/7 EOR

